// TIA Portal V17 export
// export: Created 2026-05-13T13:53:19.1488098Z, ExportSetting WithDefaults, DisplayName Totally Integrated Automation Portal, DisplayVersion V17 Update 4, DisplayName TIA Portal Openness, DisplayVersion V17 Update 4, DisplayName TIA Portal Version Control Interface, DisplayVersion V17, DisplayName SINAMICS Startdrive Advanced, DisplayVersion V17, DisplayName SINAMICS Startdrive G130, G150, S120, S150, SINAMICS MV, S210, DisplayVersion V17, DisplayName SINAMICS Startdrive G110M, G120, G120C, G120D, G120P, G115D, DisplayVersion V17, DisplayName STEP 7 Professional, DisplayVersion V17 Update 4, DisplayName STEP 7 Safety, DisplayVersion V17, DisplayName WinCC Professional, DisplayVersion V17 Update 4
VBScript "Codex_VBFunction_Loop"  Type=Sub, Comment="Codex VBS import/export loop test. Object name and Sub name must match."
  ' Codex closed-loop import/export verification.
  ' Keep the object name and the generated Sub name identical: Codex_VBFunction_Loop.
  SmartTags("Codex_VBS_Input") = "IN_OK"
  SmartTags("Codex_VBS_Output") = "OUT_OK"
